PROGRAM Data
VAR
	i					:INT; //loop index
END_VAR

// Local Time
	GVL_Status.fbLocalTime(bEnable := TRUE);	// Current Time

//Remove Total Product Data
	IF GVL_HMI.bRemoveProductData THEN
		FOR i := 0 TO cMaxStationNo DO
			astProductData[i] := astProductData[cMaxStationNo+1];
		END_FOR;
		GVL_HMI.bRemoveProductData := FALSE;
	END_IF

//Data Shift
	FOR i := 0 TO (cMaxStationNo) DO
		IF i > 0 AND i <= cMaxStationNo THEN  // 범위 체크 추가
			IF abMoveShift[i] = TRUE THEN
				astProductData[i] := astProductData[i-1];
				astProductData[i-1] := astProductData[cMaxStationNo+1]; // Delete Data before Station
				abMoveShift[i] := FALSE;
			END_IF
			
			IF abStartTimeStamp[i] AND GVL_Status.fbLocalTime.bValid THEN
				astProductData[i].dtStartTime := SYSTEMTIME_TO_DT(GVL_Status.fbLocalTime.systemTime);
			END_IF
			IF abEndTimeStamp[i] AND GVL_Status.fbLocalTime.bValid THEN
				astProductData[i].dtEndTime := SYSTEMTIME_TO_DT(GVL_Status.fbLocalTime.systemTime);
			END_IF		
			astProductData[i].tProcessTime	:= astProductData[i].dtEndTime - astProductData[i].dtStartTime;
		END_IF
	END_FOR;

END_PROGRAM

(* stored: Version 1.1.0.1
   POU Data: Id {562dac83-2e05-4857-b372-a2a336e400f8}, SpecialFunc None *)
